TYPE ST_Parameters :
STRUCT
END_STRUCT
END_TYPE

(* stored: Version 1.1.0.1, ProductVersion 3.1.4024.10
   DUT ST_Parameters: Id {4a8e0373-cad6-4939-9566-47874b160b63} *)
